PROGRAM MAIN
VAR
END_VAR

END_PROGRAM

(* stored: Version 1.1.0.1
   POU MAIN: Id {9052f2e0-61c9-4d48-84b8-36a4179fbc7c} *)
